# EPICS substitutions: vacuum/MAIN_TRUNK/vacApp/Db/l402_agilent4uhv.substitutions
# Agilent4UHV substitutions file

file db/agilent4uhv.db
{
     pattern {LOCA,			DEV,			PORT,		ADDR,	TIMEOUT}
     		{HL4,			VL402_1,		4uhv_1,		0,		0.2}
     		{HL4,			VL402_2,		4uhv_2,		0,		0.2}
}

file db/agilent4uhv_alias.db
{
     pattern {LOCA,			DEV,			SUB1,					SUB2,				SUB3,					SUB4,				PORT,		ADDR,	TIMEOUT}
     		{HL4,			VL402_1,		IP01:L402_Acc601,		IP02:L402_Acc602,	IP03:L402_Acc603,		IP04:L402_Acc604,		4uhv_1,		0,		0.2}
			{HL4,			VL402_2,		IP05:L402_Acc605,		IP06:L402_Wave601,	IP07:L402_Kly601,		IP08:Empty,			4uhv_2,		0,		0.2}
}
